VAR_GLOBAL
	
	// represents the net DC offset compensation multiplier
	XMEAS_ILOOP_CAL	: ARRAY[1..4] OF LREAL	:= 
				[
					// XMEAS tx-rx path
					0.999825, // A flow
					0.9985, // D flow
					1.0  , // E flow
					1.0001  // Reactor pressure
				];		
				
	XMV_ILOOP_CAL	: ARRAY[1..4] OF LREAL	:= 
				[
					// XMV tx-rx path
					1.00025, 	// D valve
					0.99875, 	// E valve
					1.00125, 	// A valve
					1.00075	 	// RCW Valve
				];					
END_VAR

(* stored: Version 1.1.0.1, ProductVersion 3.1.0.36
   GVL G_ICAL: Id {935515b6-9958-46e8-93f4-1544d0ed3c39} *)
